(* CODESYS project Device.Plc Logic.Application.Nivel.export

Project tree, tasks and I/O mapping:
  program Nivel [LD]
*)

// Nivel
PROGRAM Nivel
VAR
	RMISTURA_0: RMISTURA;
	Niv: REAL;
	
END_VAR

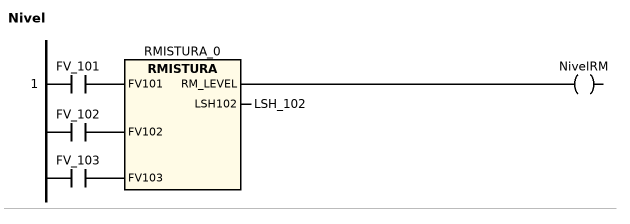
// NETWORK 1
RMISTURA_0(FV101 := FV_101, FV102 := FV_102, FV103 := FV_103, LSH102 => LSH_102); // RMISTURA
NivelRM := RMISTURA_0.RM_LEVEL;

END_PROGRAM
